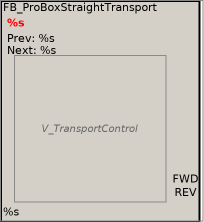
VISUALIZATION V_ProBoxStraightTransport  // 204x222
VAR_INPUT
	ZoneIx			: INT;
END_VAR

VAR_IN_OUT	
	{attribute 'VAR_IN_OUT_AS_POINTER'}
	fbFunction		: FB_ProBoxStraightTransport;		
END_VAR
    Rectangle (0,0 200x222), colour toggle: fbFunction.BaseFunctionData.ZoneOrders[ZoneIx].Drive_Run OR fbFunction.BaseFunctionData.ZoneOrders[ZoneIx].Drive_RunRev
    Label (168,172 35x14), "FWD", invisible if: NOT fbFunction.BaseFunctionData.ZoneOrders[ZoneIx].Drive_Run
    Rectangle (0,204 200x16), "%s", text variable: fbFunction.ConfigFunction.Zone[ZoneIx].ZoneName
    Label (168,183 35x19), "REV", invisible if: NOT fbFunction.BaseFunctionData.ZoneOrders[ZoneIx].Drive_RunRev
    Label (0,0 200x15), "FB_ProBoxStraightTransport"
    Rectangle (4,15 194x16), "%s", tooltip "%s", text variable: fbFunction.FunctionData.ErrorData.Error.ErrorCode.Conv, invisible if: fbFunction.FunctionData.ErrorData.ErrorState = E_ErrorState.OPERATIONAL
        p4168582468: fbFunction.FunctionData.ErrorData.Error.ErrorParam
    Frame (14,55 152x147)
        shows V_TransportControl(TransportControl := fbFunction.fbTransportControl[ZoneIx], ZoneData := fbFunction.ZoneData[ZoneIx])
    Rectangle (4,32 200x13), "Prev: %s", tooltip "FunctionInterface.in.ePrevFunctionNumber", text variable: fbFunction.FunctionInterface.In.ePrevFunctionNumber
    Rectangle (4,44 200x13), "Next: %s", tooltip "FunctionInterface.in.eNextFunctionNumber", text variable: fbFunction.FunctionInterface.In.eNextFunctionNumber
END_VISUALIZATION

(* stored: Version 1.1.0.1, ProductVersion 3.1.4024.9
   Visu V_ProBoxStraightTransport: Id {88077f12-50a3-4855-9cd8-e5d3453e2836} *)
